LIN {X 0,Y 123.721,Z 466.518,A -85,B 0,C 180,E1 5812.106,E2 5812.106} C_VEL
LIN {X 0,Y 125.333,Z 474.545,A -85,B 0,C 180,E1 5807.962,E2 5807.962} C_VEL
LIN {X 0,Y 127.051,Z 480.548,A -85,B 0,C 180,E1 5806.881,E2 5806.881} C_VEL
LIN {X 0,Y 126.719,Z 512.471,A -85,B 0,C 180,E1 5803.232,E2 5803.232} C_VEL
LIN {X 0,Y 126.942,Z 529.099,A -85,B 0,C 180,E1 5801.274,E2 5801.274} C_VEL
LIN {X 0,Y 116.275,Z 624.974,A -85,B 0,C 180,E1 5791.007,E2 5791.007} C_VEL
LIN {X 0,Y 114.11,Z 644.035,A -85,B 0,C 180,E1 5787.956,E2 5787.956} C_VEL
LIN {X 0,Y 111.654,Z 663.331,A -85,B 0,C 180,E1 5783.765,E2 5783.765} C_VEL
LIN {X 0,Y 109.356,Z 682.14,A -85,B 0,C 180,E1 5778.388,E2 5778.388} C_VEL
LIN {X 0,Y 107.675,Z 699.18,A -85,B 0,C 180,E1 5772.061,E2 5772.061} C_VEL
LIN {X 0,Y 106.977,Z 713.625,A -85,B 0,C 180,E1 5765.364,E2 5765.364} C_VEL
LIN {X 0,Y 107.37,Z 725.986,A -85,B 0,C 180,E1 5758.4,E2 5758.4} C_VEL
LIN {X 0,Y 109.143,Z 736.932,A -85,B 0,C 180,E1 5751.041,E2 5751.041} C_VEL
LIN {X 0,Y 113.112,Z 747.249,A -85,B 0,C 180,E1 5743.041,E2 5743.041} C_VEL
LIN {X 0,Y 119.26,Z 755.624,A -85,B 0,C 180,E1 5735.745,E2 5735.745} C_VEL
LIN {X 0,Y 127.977,Z 762.647,A -85,B 0,C 180,E1 5728.96,E2 5728.96} C_VEL
LIN {X 0,Y 139.113,Z 768.269,A -85,B 0,C 180,E1 5722.921,E2 5722.921} C_VEL
LIN {X 0,Y 124.03,Z 769.681,A -85,B 0,C 180,E1 5713.891,E2 5713.891} C_VEL
LIN {X 0,Y 113.887,Z 769.686,A -85,B 0,C 180,E1 5702.381,E2 5702.381} C_VEL
LIN {X 0,Y 110.648,Z 768.902,A -85,B 0,C 180,E1 5693.994,E2 5693.994} C_VEL
LIN {X 0,Y 107.857,Z 776.455,A -85,B 0,C 180,E1 5688.933,E2 5688.933} C_VEL
LIN {X 0,Y 106.873,Z 787.522,A -85,B 0,C 180,E1 5680.239,E2 5680.239} C_VEL
LIN {X 0,Y 107.326,Z 795.234,A -85,B 0,C 180,E1 5672.67,E2 5672.67} C_VEL
LIN {X 0,Y 107.583,Z 799.108,A -85,B 0,C 180,E1 5667.87,E2 5667.87} C_VEL
LIN {X 0,Y 106.675,Z 803.029,A -85,B 0,C 180,E1 5660.831,E2 5660.831} C_VEL
LIN {X 0,Y 107.675,Z 807.586,A -85,B 0,C 180,E1 5649.337,E2 5649.337} C_VEL
LIN {X 0,Y 113.967,Z 810.858,A -85,B 0,C 180,E1 5637.048,E2 5637.048} C_VEL
LIN {X 0,Y 126.113,Z 812.492,A -85,B 0,C 180,E1 5626.176,E2 5626.176} C_VEL
LIN {X 0,Y 126.877,Z 812.523,A -85,B 0,C 180,E1 5625.679,E2 5625.679} C_VEL
LIN {X 0,Y 127.463,Z 812.423,A -85,B 0,C 180,E1 5624.581,E2 5624.581} C_VEL
LIN {X 0,Y 126.538,Z 812.035,A -85,B 0,C 180,E1 5623.133,E2 5623.133} C_VEL
LIN {X 0,Y 123.586,Z 811.164,A -85,B 0,C 180,E1 5621.271,E2 5621.271} C_VEL
LIN {X 0,Y 114.796,Z 808.547,A -85,B 0,C 180,E1 5617.036,E2 5617.036} C_VEL
LIN {X 0,Y 113.804,Z 808.153,A -85,B 0,C 180,E1 5616.3,E2 5616.3} C_VEL
LIN {X 0,Y 103.814,Z 802.035,A -85,B 0,C 180,E1 5605.072,E2 5605.072} C_VEL
LIN {X 0,Y 98.87,Z 794.82,A -85,B 0,C 180,E1 5593.449,E2 5593.449} C_VEL
LIN {X 0,Y 97.448,Z 787.451,A -85,B 0,C 180,E1 5583.529,E2 5583.529} C_VEL
LIN {X 0,Y 97.238,Z 779.92,A -85,B 0,C 180,E1 5575.281,E2 5575.281} C_VEL
LIN {X 0,Y 98.022,Z 769.975,A -85,B 0,C 180,E1 5566.431,E2 5566.431} C_VEL
LIN {X 0,Y 100.32,Z 757.927,A -85,B 0,C 180,E1 5557.744,E2 5557.744} C_VEL
LIN {X 0,Y 104.103,Z 744.078,A -85,B 0,C 180,E1 5549.815,E2 5549.815} C_VEL
LIN {X 0,Y 109.128,Z 728.223,A -85,B 0,C 180,E1 5542.791,E2 5542.791} C_VEL
LIN {X 0,Y 114.606,Z 711.516,A -85,B 0,C 180,E1 5537.116,E2 5537.116} C_VEL
LIN {X 0,Y 120.618,Z 692.425,A -85,B 0,C 180,E1 5532.179,E2 5532.179} C_VEL
LIN {X 0,Y 125.944,Z 673.888,A -85,B 0,C 180,E1 5528.557,E2 5528.557} C_VEL
LIN {X 0,Y 131.132,Z 652.804,A -85,B 0,C 180,E1 5525.515,E2 5525.515} C_VEL
LIN {X 0,Y 135.576,Z 630.555,A -85,B 0,C 180,E1 5523.193,E2 5523.193} C_VEL
LIN {X 0,Y 155.35,Z 515.756,A -85,B 0,C 180,E1 5515.036,E2 5515.036} C_VEL
LIN {X 0,Y 146.72,Z 495.36,A -85,B 0,C 180,E1 5509.751,E2 5509.751} C_VEL
LIN {X 0,Y 139.149,Z 478.944,A -85,B 0,C 180,E1 5504.513,E2 5504.513} C_VEL
LIN {X 0,Y 132.05,Z 464.915,A -85,B 0,C 180,E1 5498.93,E2 5498.93} C_VEL
LIN {X 0,Y 126.321,Z 454.594,A -85,B 0,C 180,E1 5493.79,E2 5493.79} C_VEL
LIN {X 0,Y 121.035,Z 445.893,A -85,B 0,C 180,E1 5488.344,E2 5488.344} C_VEL
LIN {X 0,Y 117.879,Z 441.07,A -85,B 0,C 180,E1 5484.646,E2 5484.646} C_VEL
LIN {X 0,Y 115.952,Z 438.032,A -85,B 0,C 180,E1 5482.07,E2 5482.07} C_VEL
LIN {X 0,Y 112.145,Z 438.158,A -85,B 0,C 180,E1 5478.167,E2 5478.167} C_VEL
LIN {X 0,Y 109.969,Z 438.898,A -85,B 0,C 180,E1 5475.789,E2 5475.789} C_VEL
LIN {X 0,Y 108.87,Z 438.667,A -85,B 0,C 180,E1 5474.28,E2 5474.28} C_VEL
LIN {X 0,Y 111.114,Z 446.42,A -85,B 0,C 180,E1 5467.794,E2 5467.794} C_VEL
LIN {X 0,Y 113.434,Z 455.846,A -85,B 0,C 180,E1 5461.001,E2 5461.001} C_VEL
LIN {X 0,Y 115.802,Z 466.855,A -85,B 0,C 180,E1 5454.046,E2 5454.046} C_VEL
LIN {X 0,Y 117.31,Z 474.41,A -85,B 0,C 180,E1 5449.866,E2 5449.866} C_VEL
LIN {X 0,Y 119.728,Z 482.332,A -85,B 0,C 180,E1 5448.282,E2 5448.282} C_VEL
LIN {X 0,Y 119.282,Z 515.284,A -85,B 0,C 180,E1 5444.26,E2 5444.26} C_VEL
LIN {X 0,Y 119.355,Z 529.39,A -85,B 0,C 180,E1 5442.498,E2 5442.498} C_VEL
LIN {X 0,Y 108.536,Z 622.949,A -85,B 0,C 180,E1 5431.831,E2 5431.831} C_VEL
LIN {X 0,Y 106.255,Z 642.844,A -85,B 0,C 180,E1 5428.527,E2 5428.527} C_VEL
LIN {X 0,Y 103.774,Z 662.039,A -85,B 0,C 180,E1 5424.173,E2 5424.173} C_VEL
LIN {X 0,Y 101.618,Z 679.408,A -85,B 0,C 180,E1 5418.948,E2 5418.948} C_VEL
LIN {X 0,Y 99.948,Z 695.818,A -85,B 0,C 180,E1 5412.715,E2 5412.715} C_VEL
LIN {X 0,Y 99.177,Z 710.919,A -85,B 0,C 180,E1 5405.497,E2 5405.497} C_VEL
LIN {X 0,Y 99.552,Z 723.373,A -85,B 0,C 180,E1 5398.274,E2 5398.274} C_VEL
LIN {X 0,Y 101.704,Z 736.139,A -85,B 0,C 180,E1 5389.457,E2 5389.457} C_VEL
LIN {X 0,Y 106.251,Z 746.98,A -85,B 0,C 180,E1 5380.771,E2 5380.771} C_VEL
LIN {X 0,Y 113.993,Z 756.585,A -85,B 0,C 180,E1 5372.299,E2 5372.299} C_VEL
LIN {X 0,Y 123.628,Z 763.772,A -85,B 0,C 180,E1 5365.52,E2 5365.52} C_VEL
LIN {X 0,Y 128.584,Z 766.518,A -85,B 0,C 180,E1 5362.772,E2 5362.772} C_VEL
LIN {X 0,Y 114.403,Z 766.985,A -85,B 0,C 180,E1 5352.977,E2 5352.977} C_VEL
LIN {X 0,Y 105.299,Z 766.112,A -85,B 0,C 180,E1 5340.216,E2 5340.216} C_VEL
LIN {X 0,Y 103.59,Z 765.612,A -85,B 0,C 180,E1 5335.131,E2 5335.131} C_VEL
LIN {X 0,Y 100.37,Z 773.329,A -85,B 0,C 180,E1 5329.798,E2 5329.798} C_VEL
LIN {X 0,Y 99.169,Z 784.781,A -85,B 0,C 180,E1 5320.456,E2 5320.456} C_VEL
LIN {X 0,Y 99.688,Z 792.768,A -85,B 0,C 180,E1 5312.299,E2 5312.299} C_VEL
LIN {X 0,Y 100.047,Z 796.404,A -85,B 0,C 180,E1 5307.709,E2 5307.709} C_VEL
LIN {X 0,Y 99.083,Z 800.833,A -85,B 0,C 180,E1 5299.535,E2 5299.535} C_VEL
LIN {X 0,Y 100.78,Z 805.742,A -85,B 0,C 180,E1 5286.619,E2 5286.619} C_VEL
LIN {X 0,Y 108.267,Z 809.203,A -85,B 0,C 180,E1 5273.768,E2 5273.768} C_VEL
LIN {X 0,Y 121.516,Z 811.112,A -85,B 0,C 180,E1 5262.919,E2 5262.919} C_VEL
LIN {X 0,Y 122.391,Z 811.157,A -85,B 0,C 180,E1 5262.319,E2 5262.319} C_VEL
LIN {X 0,Y 113.804,Z 808.153,A -85,B 0,C 180,E1 5256.3,E2 5256.3} C_VEL
LIN {X 0,Y 109.274,Z 806.262,A -85,B 0,C 180,E1 5253.207,E2 5253.207} C_VEL
LIN {X 0,Y 96.639,Z 799.888,A -85,B 0,C 180,E1 5245.209,E2 5245.209} C_VEL
LIN {X 0,Y 93.598,Z 797.166,A -85,B 0,C 180,E1 5241.222,E2 5241.222} C_VEL
LIN {X 0,Y 90.215,Z 789.137,A -85,B 0,C 180,E1 5228.925,E2 5228.925} C_VEL
LIN {X 0,Y 89.552,Z 782.607,A -85,B 0,C 180,E1 5220.639,E2 5220.639} C_VEL
LIN {X 0,Y 89.61,Z 774.104,A -85,B 0,C 180,E1 5211.659,E2 5211.659} C_VEL
LIN {X 0,Y 91.062,Z 762.989,A -85,B 0,C 180,E1 5202.094,E2 5202.094} C_VEL
LIN {X 0,Y 94.319,Z 749.505,A -85,B 0,C 180,E1 5192.881,E2 5192.881} C_VEL
LIN {X 0,Y 99.036,Z 734.325,A -85,B 0,C 180,E1 5184.863,E2 5184.863} C_VEL
LIN {X 0,Y 104.744,Z 717.443,A -85,B 0,C 180,E1 5178.07,E2 5178.07} C_VEL
LIN {X 0,Y 110.762,Z 699.456,A -85,B 0,C 180,E1 5172.612,E2 5172.612} C_VEL
LIN {X 0,Y 116.626,Z 680.494,A -85,B 0,C 180,E1 5168.329,E2 5168.329} C_VEL
LIN {X 0,Y 122.369,Z 659.306,A -85,B 0,C 180,E1 5164.797,E2 5164.797} C_VEL
LIN {X 0,Y 127.131,Z 637.978,A -85,B 0,C 180,E1 5162.224,E2 5162.224} C_VEL
LIN {X 0,Y 145.128,Z 537.776,A -85,B 0,C 180,E1 5154.544,E2 5154.544} C_VEL
LIN {X 0,Y 148.695,Z 518.047,A -85,B 0,C 180,E1 5153.269,E2 5153.269} C_VEL
LIN {X 0,Y 140.634,Z 498.608,A -85,B 0,C 180,E1 5147.908,E2 5147.908} C_VEL
LIN {X 0,Y 133.872,Z 483.562,A -85,B 0,C 180,E1 5142.838,E2 5142.838} C_VEL
LIN {X 0,Y 127.212,Z 469.981,A -85,B 0,C 180,E1 5137.162,E2 5137.162} C_VEL
LIN {X 0,Y 121.883,Z 460.1,A -85,B 0,C 180,E1 5131.946,E2 5131.946} C_VEL
LIN {X 0,Y 117.073,Z 451.938,A -85,B 0,C 180,E1 5126.573,E2 5126.573} C_VEL
LIN {X 0,Y 114.17,Z 447.292,A -85,B 0,C 180,E1 5122.831,E2 5122.831} C_VEL
LIN {X 0,Y 113.07,Z 445.717,A -85,B 0,C 180,E1 5121.354,E2 5121.354} C_VEL
LIN {X 0,Y 110.544,Z 446.078,A -85,B 0,C 180,E1 5118.786,E2 5118.786} C_VEL
LIN {X 0,Y 107.633,Z 446.625,A -85,B 0,C 180,E1 5115.474,E2 5115.474} C_VEL
LIN {X 0,Y 104.899,Z 448.123,A -85,B 0,C 180,E1 5112.241,E2 5112.241} C_VEL
LIN {X 0,Y 103.67,Z 448.229,A -85,B 0,C 180,E1 5110.124,E2 5110.124} C_VEL
LIN {X 0,Y 105.846,Z 457.247,A -85,B 0,C 180,E1 5103.036,E2 5103.036} C_VEL
LIN {X 0,Y 108.015,Z 467.637,A -85,B 0,C 180,E1 5095.942,E2 5095.942} C_VEL
LIN {X 0,Y 109.337,Z 474.358,A -85,B 0,C 180,E1 5091.966,E2 5091.966} C_VEL
LIN {X 0,Y 112.418,Z 484.295,A -85,B 0,C 180,E1 5089.775,E2 5089.775} C_VEL
LIN {X 0,Y 111.853,Z 518.434,A -85,B 0,C 180,E1 5085.323,E2 5085.323} C_VEL
LIN {X 0,Y 111.808,Z 529.579,A -85,B 0,C 180,E1 5083.851,E2 5083.851} C_VEL
LIN {X 0,Y 100.23,Z 626.422,A -85,B 0,C 180,E1 5071.919,E2 5071.919} C_VEL
LIN {X 0,Y 97.916,Z 645.376,A -85,B 0,C 180,E1 5068.349,E2 5068.349} C_VEL
LIN {X 0,Y 95.286,Z 665.471,A -85,B 0,C 180,E1 5063.173,E2 5063.173} C_VEL
LIN {X 0,Y 93.159,Z 683.027,A -85,B 0,C 180,E1 5057.209,E2 5057.209} C_VEL
LIN {X 0,Y 91.742,Z 699.415,A -85,B 0,C 180,E1 5050.043,E2 5050.043} C_VEL
LIN {X 0,Y 91.405,Z 712.924,A -85,B 0,C 180,E1 5042.822,E2 5042.822} C_VEL
LIN {X 0,Y 92.524,Z 726.836,A -85,B 0,C 180,E1 5033.797,E2 5033.797} C_VEL
LIN {X 0,Y 95.591,Z 738.612,A -85,B 0,C 180,E1 5024.842,E2 5024.842} C_VEL
LIN {X 0,Y 102.11,Z 750.1,A -85,B 0,C 180,E1 5015.1,E2 5015.1} C_VEL
LIN {X 0,Y 111.506,Z 759.323,A -85,B 0,C 180,E1 5006.841,E2 5006.841} C_VEL
LIN {X 0,Y 118.345,Z 763.963,A -85,B 0,C 180,E1 5002.534,E2 5002.534} C_VEL
LIN {X 0,Y 104.148,Z 763.568,A -85,B 0,C 180,E1 4990.755,E2 4990.755} C_VEL
LIN {X 0,Y 96.875,Z 761.886,A -85,B 0,C 180,E1 4976.678,E2 4976.678} C_VEL
LIN {X 0,Y 93.002,Z 769.991,A -85,B 0,C 180,E1 4970.78,E2 4970.78} C_VEL
LIN {X 0,Y 91.512,Z 782.027,A -85,B 0,C 180,E1 4960.478,E2 4960.478} C_VEL
LIN {X 0,Y 92.092,Z 790.143,A -85,B 0,C 180,E1 4951.867,E2 4951.867} C_VEL
LIN {X 0,Y 92.515,Z 793.931,A -85,B 0,C 180,E1 4946.902,E2 4946.902} C_VEL
LIN {X 0,Y 91.623,Z 798.409,A -85,B 0,C 180,E1 4938.033,E2 4938.033} C_VEL
LIN {X 0,Y 93.946,Z 803.567,A -85,B 0,C 180,E1 4924.128,E2 4924.128} C_VEL
LIN {X 0,Y 102.499,Z 807.357,A -85,B 0,C 180,E1 4910.649,E2 4910.649} C_VEL
LIN {X 0,Y 112.424,Z 809.109,A -85,B 0,C 180,E1 4902.424,E2 4902.424} C_VEL
LIN {X 0,Y 99.893,Z 803.047,A -85,B 0,C 180,E1 4891.364,E2 4891.364} C_VEL
LIN {X 0,Y 93.598,Z 797.166,A -85,B 0,C 180,E1 4881.222,E2 4881.222} C_VEL
LIN {X 0,Y 91.082,Z 794.298,A -85,B 0,C 180,E1 4877.067,E2 4877.067} C_VEL
LIN {X 0,Y 85.995,Z 788.825,A -85,B 0,C 180,E1 4870.746,E2 4870.746} C_VEL
LIN {X 0,Y 82.222,Z 782.653,A -85,B 0,C 180,E1 4863.824,E2 4863.824} C_VEL
LIN {X 0,Y 81.888,Z 780.974,A -85,B 0,C 180,E1 4861.77,E2 4861.77} C_VEL
LIN {X 0,Y 81.828,Z 772.489,A -85,B 0,C 180,E1 4852.275,E2 4852.275} C_VEL
LIN {X 0,Y 83.277,Z 761.101,A -85,B 0,C 180,E1 4841.809,E2 4841.809} C_VEL
LIN {X 0,Y 86.73,Z 747.302,A -85,B 0,C 180,E1 4831.792,E2 4831.792} C_VEL
LIN {X 0,Y 91.77,Z 731.804,A -85,B 0,C 180,E1 4823.183,E2 4823.183} C_VEL
LIN {X 0,Y 97.734,Z 714.838,A -85,B 0,C 180,E1 4816.143,E2 4816.143} C_VEL
LIN {X 0,Y 103.978,Z 696.725,A -85,B 0,C 180,E1 4810.564,E2 4810.564} C_VEL
LIN {X 0,Y 110.169,Z 677.178,A -85,B 0,C 180,E1 4806.124,E2 4806.124} C_VEL
LIN {X 0,Y 115.848,Z 656.61,A -85,B 0,C 180,E1 4802.699,E2 4802.699} C_VEL
LIN {X 0,Y 120.749,Z 634.715,A -85,B 0,C 180,E1 4800.11,E2 4800.11} C_VEL
LIN {X 0,Y 142.151,Z 520.396,A -85,B 0,C 180,E1 4791.4,E2 4791.4} C_VEL
LIN {X 0,Y 134.468,Z 501.434,A -85,B 0,C 180,E1 4785.803,E2 4785.803} C_VEL
LIN {X 0,Y 127.943,Z 486.588,A -85,B 0,C 180,E1 4780.429,E2 4780.429} C_VEL
LIN {X 0,Y 121.851,Z 473.881,A -85,B 0,C 180,E1 4774.707,E2 4774.707} C_VEL
LIN {X 0,Y 116.348,Z 463.379,A -85,B 0,C 180,E1 4768.646,E2 4768.646} C_VEL
LIN {X 0,Y 111.637,Z 455.203,A -85,B 0,C 180,E1 4762.538,E2 4762.538} C_VEL
LIN {X 0,Y 110.391,Z 453.587,A -85,B 0,C 180,E1 4760.849,E2 4760.849} C_VEL
LIN {X 0,Y 105.65,Z 454.774,A -85,B 0,C 180,E1 4755.755,E2 4755.755} C_VEL
LIN {X 0,Y 102.852,Z 455.957,A -85,B 0,C 180,E1 4752.308,E2 4752.308} C_VEL
LIN {X 0,Y 101.988,Z 456.324,A -85,B 0,C 180,E1 4751.124,E2 4751.124} C_VEL
LIN {X 0,Y 99.384,Z 458.401,A -85,B 0,C 180,E1 4747.523,E2 4747.523} C_VEL
LIN {X 0,Y 98.286,Z 458.631,A -85,B 0,C 180,E1 4745.349,E2 4745.349} C_VEL
LIN {X 0,Y 100.3,Z 468.623,A -85,B 0,C 180,E1 4737.925,E2 4737.925} C_VEL
LIN {X 0,Y 101.387,Z 474.232,A -85,B 0,C 180,E1 4734.332,E2 4734.332} C_VEL
LIN {X 0,Y 105.158,Z 486.038,A -85,B 0,C 180,E1 4731.45,E2 4731.45} C_VEL
LIN {X 0,Y 104.426,Z 521.241,A -85,B 0,C 180,E1 4726.525,E2 4726.525} C_VEL
LIN {X 0,Y 104.26,Z 529.903,A -85,B 0,C 180,E1 4725.316,E2 4725.316} C_VEL
LIN {X 0,Y 92.313,Z 625.986,A -85,B 0,C 180,E1 4712.56,E2 4712.56} C_VEL
LIN {X 0,Y 89.751,Z 646.386,A -85,B 0,C 180,E1 4708.41,E2 4708.41} C_VEL
LIN {X 0,Y 87.193,Z 665.725,A -85,B 0,C 180,E1 4702.948,E2 4702.948} C_VEL
LIN {X 0,Y 85.022,Z 684.07,A -85,B 0,C 180,E1 4696.044,E2 4696.044} C_VEL
LIN {X 0,Y 83.846,Z 699.623,A -85,B 0,C 180,E1 4688.573,E2 4688.573} C_VEL
LIN {X 0,Y 83.83,Z 714.169,A -85,B 0,C 180,E1 4680.001,E2 4680.001} C_VEL
LIN {X 0,Y 85.319,Z 726.551,A -85,B 0,C 180,E1 4671.238,E2 4671.238} C_VEL
LIN {X 0,Y 89.029,Z 738.457,A -85,B 0,C 180,E1 4661.673,E2 4661.673} C_VEL
LIN {X 0,Y 95.494,Z 748.999,A -85,B 0,C 180,E1 4652.569,E2 4652.569} C_VEL
LIN {X 0,Y 104.93,Z 758.162,A -85,B 0,C 180,E1 4644.462,E2 4644.462} C_VEL
LIN {X 0,Y 108.323,Z 760.799,A -85,B 0,C 180,E1 4642.111,E2 4642.111} C_VEL
LIN {X 0,Y 95.171,Z 759.575,A -85,B 0,C 180,E1 4629.077,E2 4629.077} C_VEL
LIN {X 0,Y 90.239,Z 758.073,A -85,B 0,C 180,E1 4618.273,E2 4618.273} C_VEL
LIN {X 0,Y 86.024,Z 765.743,A -85,B 0,C 180,E1 4612.554,E2 4612.554} C_VEL
LIN {X 0,Y 83.939,Z 776.554,A -85,B 0,C 180,E1 4603.081,E2 4603.081} C_VEL
LIN {X 0,Y 84.274,Z 785.664,A -85,B 0,C 180,E1 4593.401,E2 4593.401} C_VEL
LIN {X 0,Y 85.113,Z 790.885,A -85,B 0,C 180,E1 4586.633,E2 4586.633} C_VEL
LIN {X 0,Y 84.257,Z 795.604,A -85,B 0,C 180,E1 4576.969,E2 4576.969} C_VEL
LIN {X 0,Y 87.097,Z 801.024,A -85,B 0,C 180,E1 4561.922,E2 4561.922} C_VEL
LIN {X 0,Y 97.124,Z 805.268,A -85,B 0,C 180,E1 4547.199,E2 4547.199} C_VEL
LIN {X 0,Y 102.565,Z 806.461,A -85,B 0,C 180,E1 4542.46,E2 4542.46} C_VEL
LIN {X 0,Y 90.222,Z 799.306,A -85,B 0,C 180,E1 4529.913,E2 4529.913} C_VEL
LIN {X 0,Y 83.846,Z 790.967,A -85,B 0,C 180,E1 4515.918,E2 4515.918} C_VEL
LIN {X 0,Y 82.11,Z 783.382,A -85,B 0,C 180,E1 4504.889,E2 4504.889} C_VEL
LIN {X 0,Y 81.888,Z 780.974,A -85,B 0,C 180,E1 4501.77,E2 4501.77} C_VEL
LIN {X 0,Y 81.018,Z 777.486,A -85,B 0,C 180,E1 4497.857,E2 4497.857} C_VEL
LIN {X 0,Y 78.361,Z 771.552,A -85,B 0,C 180,E1 4492.363,E2 4492.363} C_VEL
LIN {X 0,Y 75.4,Z 762.922,A -85,B 0,C 180,E1 4484.847,E2 4484.847} C_VEL
LIN {X 0,Y 75.493,Z 759.219,A -85,B 0,C 180,E1 4481.571,E2 4481.571} C_VEL
LIN {X 0,Y 78.882,Z 745.991,A -85,B 0,C 180,E1 4471.205,E2 4471.205} C_VEL
LIN {X 0,Y 84.18,Z 730.279,A -85,B 0,C 180,E1 4461.855,E2 4461.855} C_VEL
LIN {X 0,Y 90.363,Z 713.341,A -85,B 0,C 180,E1 4454.463,E2 4454.463} C_VEL
LIN {X 0,Y 97.067,Z 694.602,A -85,B 0,C 180,E1 4448.476,E2 4448.476} C_VEL
LIN {X 0,Y 103.57,Z 674.696,A -85,B 0,C 180,E1 4443.875,E2 4443.875} C_VEL
LIN {X 0,Y 109.519,Z 653.453,A -85,B 0,C 180,E1 4440.373,E2 4440.373} C_VEL
LIN {X 0,Y 114.494,Z 631.417,A -85,B 0,C 180,E1 4437.811,E2 4437.811} C_VEL
LIN {X 0,Y 135.589,Z 522.526,A -85,B 0,C 180,E1 4429.324,E2 4429.324} C_VEL
LIN {X 0,Y 128.396,Z 504.331,A -85,B 0,C 180,E1 4423.573,E2 4423.573} C_VEL
LIN {X 0,Y 122.113,Z 489.542,A -85,B 0,C 180,E1 4417.796,E2 4417.796} C_VEL
LIN {X 0,Y 116.23,Z 476.958,A -85,B 0,C 180,E1 4411.602,E2 4411.602} C_VEL
LIN {X 0,Y 110.768,Z 466.31,A -85,B 0,C 180,E1 4404.691,E2 4404.691} C_VEL
LIN {X 0,Y 108.029,Z 461.515,A -85,B 0,C 180,E1 4400.679,E2 4400.679} C_VEL
LIN {X 0,Y 104.264,Z 462.552,A -85,B 0,C 180,E1 4396.694,E2 4396.694} C_VEL
LIN {X 0,Y 100.714,Z 464.062,A -85,B 0,C 180,E1 4392.378,E2 4392.378} C_VEL
LIN {X 0,Y 97.805,Z 466.095,A -85,B 0,C 180,E1 4388.406,E2 4388.406} C_VEL
LIN {X 0,Y 96.699,Z 466.726,A -85,B 0,C 180,E1 4386.589,E2 4386.589} C_VEL
LIN {X 0,Y 94.001,Z 469.898,A -85,B 0,C 180,E1 4382.249,E2 4382.249} C_VEL
LIN {X 0,Y 92.834,Z 470.83,A -85,B 0,C 180,E1 4379.23,E2 4379.23} C_VEL
LIN {X 0,Y 93.482,Z 474.123,A -85,B 0,C 180,E1 4377.033,E2 4377.033} C_VEL
LIN {X 0,Y 97.927,Z 487.871,A -85,B 0,C 180,E1 4373.276,E2 4373.276} C_VEL
LIN {X 0,Y 97.007,Z 524.973,A -85,B 0,C 180,E1 4367.689,E2 4367.689} C_VEL
LIN {X 0,Y 96.664,Z 530.708,A -85,B 0,C 180,E1 4366.877,E2 4366.877} C_VEL
LIN {X 0,Y 84.165,Z 627.528,A -85,B 0,C 180,E1 4352.898,E2 4352.898} C_VEL
LIN {X 0,Y 81.651,Z 646.801,A -85,B 0,C 180,E1 4348.528,E2 4348.528} C_VEL
LIN {X 0,Y 79.007,Z 666.672,A -85,B 0,C 180,E1 4342.313,E2 4342.313} C_VEL
LIN {X 0,Y 77.022,Z 684.046,A -85,B 0,C 180,E1 4335.049,E2 4335.049} C_VEL
LIN {X 0,Y 76.041,Z 699.625,A -85,B 0,C 180,E1 4326.797,E2 4326.797} C_VEL
LIN {X 0,Y 76.366,Z 713.602,A -85,B 0,C 180,E1 4317.75,E2 4317.75} C_VEL
LIN {X 0,Y 78.317,Z 726.203,A -85,B 0,C 180,E1 4308.214,E2 4308.214} C_VEL
LIN {X 0,Y 83.182,Z 738.924,A -85,B 0,C 180,E1 4297.379,E2 4297.379} C_VEL
LIN {X 0,Y 91.282,Z 750.114,A -85,B 0,C 180,E1 4287.54,E2 4287.54} C_VEL
LIN {X 0,Y 98.67,Z 756.927,A -85,B 0,C 180,E1 4281.541,E2 4281.541} C_VEL
LIN {X 0,Y 86.238,Z 754.891,A -85,B 0,C 180,E1 4266.25,E2 4266.25} C_VEL
LIN {X 0,Y 83.89,Z 753.99,A -85,B 0,C 180,E1 4260.236,E2 4260.236} C_VEL
LIN {X 0,Y 79.275,Z 761.328,A -85,B 0,C 180,E1 4254.596,E2 4254.596} C_VEL
LIN {X 0,Y 76.54,Z 770.847,A -85,B 0,C 180,E1 4245.922,E2 4245.922} C_VEL
LIN {X 0,Y 76.498,Z 780.779,A -85,B 0,C 180,E1 4235.25,E2 4235.25} C_VEL
LIN {X 0,Y 77.704,Z 787.693,A -85,B 0,C 180,E1 4226.311,E2 4226.311} C_VEL
LIN {X 0,Y 77.01,Z 791.977,A -85,B 0,C 180,E1 4217.249,E2 4217.249} C_VEL
LIN {X 0,Y 79.877,Z 797.867,A -85,B 0,C 180,E1 4200.779,E2 4200.779} C_VEL
LIN {X 0,Y 90.361,Z 802.559,A -85,B 0,C 180,E1 4185.085,E2 4185.085} C_VEL
LIN {X 0,Y 92.988,Z 803.281,A -85,B 0,C 180,E1 4182.641,E2 4182.641} C_VEL
LIN {X 0,Y 81.109,Z 795.266,A -85,B 0,C 180,E1 4168.735,E2 4168.735} C_VEL
LIN {X 0,Y 75.617,Z 786.418,A -85,B 0,C 180,E1 4153.768,E2 4153.768} C_VEL
LIN {X 0,Y 74.306,Z 778.93,A -85,B 0,C 180,E1 4142.893,E2 4142.893} C_VEL
LIN {X 0,Y 74.079,Z 770.779,A -85,B 0,C 180,E1 4133.022,E2 4133.022} C_VEL
LIN {X 0,Y 75.493,Z 759.219,A -85,B 0,C 180,E1 4121.571,E2 4121.571} C_VEL
LIN {X 0,Y 75.65,Z 753.984,A -85,B 0,C 180,E1 4117.24,E2 4117.24} C_VEL
LIN {X 0,Y 74.166,Z 744.301,A -85,B 0,C 180,E1 4110.222,E2 4110.222} C_VEL
LIN {X 0,Y 74.076,Z 736.656,A -85,B 0,C 180,E1 4105.087,E2 4105.087} C_VEL
LIN {X 0,Y 74.941,Z 733.22,A -85,B 0,C 180,E1 4102.951,E2 4102.951} C_VEL
LIN {X 0,Y 81.259,Z 716.528,A -85,B 0,C 180,E1 4094.464,E2 4094.464} C_VEL
LIN {X 0,Y 88.1,Z 698.388,A -85,B 0,C 180,E1 4087.876,E2 4087.876} C_VEL
LIN {X 0,Y 95.059,Z 678.413,A -85,B 0,C 180,E1 4082.703,E2 4082.703} C_VEL
LIN {X 0,Y 101.268,Z 657.994,A -85,B 0,C 180,E1 4078.934,E2 4078.934} C_VEL
LIN {X 0,Y 106.692,Z 635.926,A -85,B 0,C 180,E1 4076.113,E2 4076.113} C_VEL
LIN {X 0,Y 129.29,Z 525.084,A -85,B 0,C 180,E1 4067.206,E2 4067.206} C_VEL
LIN {X 0,Y 122.453,Z 507.2,A -85,B 0,C 180,E1 4061.17,E2 4061.17} C_VEL
LIN {X 0,Y 116.584,Z 492.994,A -85,B 0,C 180,E1 4055.142,E2 4055.142} C_VEL
LIN {X 0,Y 111.623,Z 481.965,A -85,B 0,C 180,E1 4049.294,E2 4049.294} C_VEL
LIN {X 0,Y 107.035,Z 472.552,A -85,B 0,C 180,E1 4042.89,E2 4042.89} C_VEL
LIN {X 0,Y 105.47,Z 469.603,A -85,B 0,C 180,E1 4040.378,E2 4040.378} C_VEL
LIN {X 0,Y 102.881,Z 470.299,A -85,B 0,C 180,E1 4037.654,E2 4037.654} C_VEL
LIN {X 0,Y 99.296,Z 471.895,A -85,B 0,C 180,E1 4033.458,E2 4033.458} C_VEL
LIN {X 0,Y 95.383,Z 474.453,A -85,B 0,C 180,E1 4028.082,E2 4028.082} C_VEL
LIN {X 0,Y 92.384,Z 477.586,A -85,B 0,C 180,E1 4023.311,E2 4023.311} C_VEL
LIN {X 0,Y 91.234,Z 478.654,A -85,B 0,C 180,E1 4020.929,E2 4020.929} C_VEL
LIN {X 0,Y 89.394,Z 482.633,A -85,B 0,C 180,E1 4018.219,E2 4018.219} C_VEL
LIN {X 0,Y 88.994,Z 483.763,A -85,B 0,C 180,E1 4017.029,E2 4017.029} C_VEL
LIN {X 0,Y 90.735,Z 490.079,A -85,B 0,C 180,E1 4015.279,E2 4015.279} C_VEL
LIN {X 0,Y 89.331,Z 530.129,A -85,B 0,C 180,E1 4008.818,E2 4008.818} C_VEL
LIN {X 0,Y 76.063,Z 628.474,A -85,B 0,C 180,E1 3993.306,E2 3993.306} C_VEL
LIN {X 0,Y 73.465,Z 647.791,A -85,B 0,C 180,E1 3988.449,E2 3988.449} C_VEL
LIN {X 0,Y 70.861,Z 667.353,A -85,B 0,C 180,E1 3981.523,E2 3981.523} C_VEL
LIN {X 0,Y 68.89,Z 686.196,A -85,B 0,C 180,E1 3972.576,E2 3972.576} C_VEL
LIN {X 0,Y 68.368,Z 701.323,A -85,B 0,C 180,E1 3963.355,E2 3963.355} C_VEL
LIN {X 0,Y 69.404,Z 715.573,A -85,B 0,C 180,E1 3952.967,E2 3952.967} C_VEL
LIN {X 0,Y 72.796,Z 729.076,A -85,B 0,C 180,E1 3941.586,E2 3941.586} C_VEL
LIN {X 0,Y 79.827,Z 742.098,A -85,B 0,C 180,E1 3929.934,E2 3929.934} C_VEL
LIN {X 0,Y 89.383,Z 752.538,A -85,B 0,C 180,E1 3920.773,E2 3920.773} C_VEL
LIN {X 0,Y 78.157,Z 749.724,A -85,B 0,C 180,E1 3903.374,E2 3903.374} C_VEL
LIN {X 0,Y 77.776,Z 749.693,A -85,B 0,C 180,E1 3902.461,E2 3902.461} C_VEL
LIN {X 0,Y 72.816,Z 756.642,A -85,B 0,C 180,E1 3896.945,E2 3896.945} C_VEL
LIN {X 0,Y 69.361,Z 765.595,A -85,B 0,C 180,E1 3888.49,E2 3888.49} C_VEL
LIN {X 0,Y 68.88,Z 776.874,A -85,B 0,C 180,E1 3875.832,E2 3875.832} C_VEL
LIN {X 0,Y 70.408,Z 784.699,A -85,B 0,C 180,E1 3865.112,E2 3865.112} C_VEL
LIN {X 0,Y 69.876,Z 789.052,A -85,B 0,C 180,E1 3855.074,E2 3855.074} C_VEL
LIN {X 0,Y 74.075,Z 795.388,A -85,B 0,C 180,E1 3836.398,E2 3836.398} C_VEL
LIN {X 0,Y 83.542,Z 799.491,A -85,B 0,C 180,E1 3822.804,E2 3822.804} C_VEL
LIN {X 0,Y 72.511,Z 791.042,A -85,B 0,C 180,E1 3807.957,E2 3807.957} C_VEL
LIN {X 0,Y 67.808,Z 782.318,A -85,B 0,C 180,E1 3792.777,E2 3792.777} C_VEL
LIN {X 0,Y 66.659,Z 775.559,A -85,B 0,C 180,E1 3782.578,E2 3782.578} C_VEL
LIN {X 0,Y 66.484,Z 766.656,A -85,B 0,C 180,E1 3771.349,E2 3771.349} C_VEL
LIN {X 0,Y 68.382,Z 754.22,A -85,B 0,C 180,E1 3758.558,E2 3758.558} C_VEL
LIN {X 0,Y 72.634,Z 739.743,A -85,B 0,C 180,E1 3747.11,E2 3747.11} C_VEL
LIN {X 0,Y 74.941,Z 733.22,A -85,B 0,C 180,E1 3742.951,E2 3742.951} C_VEL
LIN {X 0,Y 76.193,Z 727.143,A -85,B 0,C 180,E1 3739.421,E2 3739.421} C_VEL
LIN {X 0,Y 76.383,Z 713.469,A -85,B 0,C 180,E1 3732.091,E2 3732.091} C_VEL
LIN {X 0,Y 77.636,Z 705.905,A -85,B 0,C 180,E1 3728.659,E2 3728.659} C_VEL
LIN {X 0,Y 78.297,Z 703.986,A -85,B 0,C 180,E1 3727.928,E2 3727.928} C_VEL
LIN {X 0,Y 85.53,Z 684.851,A -85,B 0,C 180,E1 3722.054,E2 3722.054} C_VEL
LIN {X 0,Y 92.154,Z 665.009,A -85,B 0,C 180,E1 3717.81,E2 3717.81} C_VEL
LIN {X 0,Y 98.137,Z 643.486,A -85,B 0,C 180,E1 3714.587,E2 3714.587} C_VEL
LIN {X 0,Y 105.014,Z 611.799,A -85,B 0,C 180,E1 3711.36,E2 3711.36} C_VEL
LIN {X 0,Y 122.943,Z 527.227,A -85,B 0,C 180,E1 3704.783,E2 3704.783} C_VEL
LIN {X 0,Y 116.417,Z 509.537,A -85,B 0,C 180,E1 3698.333,E2 3698.333} C_VEL
LIN {X 0,Y 110.885,Z 495.637,A -85,B 0,C 180,E1 3691.873,E2 3691.873} C_VEL
LIN {X 0,Y 106.366,Z 485.172,A -85,B 0,C 180,E1 3685.687,E2 3685.687} C_VEL
LIN {X 0,Y 102.71,Z 477.567,A -85,B 0,C 180,E1 3679.829,E2 3679.829} C_VEL
LIN {X 0,Y 98.152,Z 479.522,A -85,B 0,C 180,E1 3674.812,E2 3674.812} C_VEL
LIN {X 0,Y 94.295,Z 481.971,A -85,B 0,C 180,E1 3669.789,E2 3669.789} C_VEL
LIN {X 0,Y 90.848,Z 485.226,A -85,B 0,C 180,E1 3664.488,E2 3664.488} C_VEL
LIN {X 0,Y 90.279,Z 485.976,A -85,B 0,C 180,E1 3663.602,E2 3663.602} C_VEL
LIN {X 0,Y 88.23,Z 489.907,A -85,B 0,C 180,E1 3660.764,E2 3660.764} C_VEL
LIN {X 0,Y 86.957,Z 493.361,A -85,B 0,C 180,E1 3659.504,E2 3659.504} C_VEL
LIN {X 0,Y 83.896,Z 502.205,A -85,B 0,C 180,E1 3656.819,E2 3656.819} C_VEL
LIN {X 0,Y 82.806,Z 505.573,A -85,B 0,C 180,E1 3655.29,E2 3655.29} C_VEL
LIN {X 0,Y 81.955,Z 530.078,A -85,B 0,C 180,E1 3650.921,E2 3650.921} C_VEL
LIN {X 0,Y 68.112,Z 628.15,A -85,B 0,C 180,E1 3634.034,E2 3634.034} C_VEL
LIN {X 0,Y 65.329,Z 648.28,A -85,B 0,C 180,E1 3628.325,E2 3628.325} C_VEL
LIN {X 0,Y 62.747,Z 667.856,A -85,B 0,C 180,E1 3620.523,E2 3620.523} C_VEL
LIN {X 0,Y 61.119,Z 684.923,A -85,B 0,C 180,E1 3611.322,E2 3611.322} C_VEL
LIN {X 0,Y 60.852,Z 700.406,A -85,B 0,C 180,E1 3600.943,E2 3600.943} C_VEL
LIN {X 0,Y 62.578,Z 715.186,A -85,B 0,C 180,E1 3588.947,E2 3588.947} C_VEL
LIN {X 0,Y 66.739,Z 728.344,A -85,B 0,C 180,E1 3577.076,E2 3577.076} C_VEL
LIN {X 0,Y 73.824,Z 740.101,A -85,B 0,C 180,E1 3566.27,E2 3566.27} C_VEL
LIN {X 0,Y 80.515,Z 747.565,A -85,B 0,C 180,E1 3559.779,E2 3559.779} C_VEL
LIN {X 0,Y 72.1,Z 745.036,A -85,B 0,C 180,E1 3545.136,E2 3545.136} C_VEL
LIN {X 0,Y 66.629,Z 751.824,A -85,B 0,C 180,E1 3539.684,E2 3539.684} C_VEL
LIN {X 0,Y 62.101,Z 761.699,A -85,B 0,C 180,E1 3529.762,E2 3529.762} C_VEL
LIN {X 0,Y 61.456,Z 774.051,A -85,B 0,C 180,E1 3514.666,E2 3514.666} C_VEL
LIN {X 0,Y 63.206,Z 781.852,A -85,B 0,C 180,E1 3503.186,E2 3503.186} C_VEL
LIN {X 0,Y 63.698,Z 788.191,A -85,B 0,C 180,E1 3485.913,E2 3485.913} C_VEL
LIN {X 0,Y 72.144,Z 794.377,A -85,B 0,C 180,E1 3466.11,E2 3466.11} C_VEL
LIN {X 0,Y 74.33,Z 795.204,A -85,B 0,C 180,E1 3463.052,E2 3463.052} C_VEL
LIN {X 0,Y 63.698,Z 785.836,A -85,B 0,C 180,E1 3446.071,E2 3446.071} C_VEL
LIN {X 0,Y 59.936,Z 777.233,A -85,B 0,C 180,E1 3430.573,E2 3430.573} C_VEL
LIN {X 0,Y 58.872,Z 769.628,A -85,B 0,C 180,E1 3419.026,E2 3419.026} C_VEL
LIN {X 0,Y 59.232,Z 759.734,A -85,B 0,C 180,E1 3406.329,E2 3406.329} C_VEL
LIN {X 0,Y 62.19,Z 746.447,A -85,B 0,C 180,E1 3392.727,E2 3392.727} C_VEL
LIN {X 0,Y 67.466,Z 731.259,A -85,B 0,C 180,E1 3381.208,E2 3381.208} C_VEL
LIN {X 0,Y 74.159,Z 714.372,A -85,B 0,C 180,E1 3372.135,E2 3372.135} C_VEL
LIN {X 0,Y 78.297,Z 703.986,A -85,B 0,C 180,E1 3367.928,E2 3367.928} C_VEL
LIN {X 0,Y 79.961,Z 697.284,A -85,B 0,C 180,E1 3365.367,E2 3365.367} C_VEL
LIN {X 0,Y 81.208,Z 678.536,A -85,B 0,C 180,E1 3358.294,E2 3358.294} C_VEL
LIN {X 0,Y 82.686,Z 672.39,A -85,B 0,C 180,E1 3356.682,E2 3356.682} C_VEL
LIN {X 0,Y 89.32,Z 651.279,A -85,B 0,C 180,E1 3352.967,E2 3352.967} C_VEL
LIN {X 0,Y 95.072,Z 628.181,A -85,B 0,C 180,E1 3350.229,E2 3350.229} C_VEL
LIN {X 0,Y 116.803,Z 529.586,A -85,B 0,C 180,E1 3342.229,E2 3342.229} C_VEL
LIN {X 0,Y 110.764,Z 512.531,A -85,B 0,C 180,E1 3335.504,E2 3335.504} C_VEL
LIN {X 0,Y 105.881,Z 499.542,A -85,B 0,C 180,E1 3328.992,E2 3328.992} C_VEL
LIN {X 0,Y 101.951,Z 489.947,A -85,B 0,C 180,E1 3322.817,E2 3322.817} C_VEL
LIN {X 0,Y 100.11,Z 485.795,A -85,B 0,C 180,E1 3319.537,E2 3319.537} C_VEL
LIN {X 0,Y 96.698,Z 487.363,A -85,B 0,C 180,E1 3315.796,E2 3315.796} C_VEL
LIN {X 0,Y 93.309,Z 489.435,A -85,B 0,C 180,E1 3311.572,E2 3311.572} C_VEL
LIN {X 0,Y 89.618,Z 492.908,A -85,B 0,C 180,E1 3306.368,E2 3306.368} C_VEL
LIN {X 0,Y 87.98,Z 495.911,A -85,B 0,C 180,E1 3304.431,E2 3304.431} C_VEL
LIN {X 0,Y 84.341,Z 505.672,A -85,B 0,C 180,E1 3301.749,E2 3301.749} C_VEL
LIN {X 0,Y 82.822,Z 509.668,A -85,B 0,C 180,E1 3300.282,E2 3300.282} C_VEL
LIN {X 0,Y 78.469,Z 522.921,A -85,B 0,C 180,E1 3297.33,E2 3297.33} C_VEL
LIN {X 0,Y 75.773,Z 531.128,A -85,B 0,C 180,E1 3294.628,E2 3294.628} C_VEL
LIN {X 0,Y 72.538,Z 542.204,A -85,B 0,C 180,E1 3291.587,E2 3291.587} C_VEL
LIN {X 0,Y 59.811,Z 630.351,A -85,B 0,C 180,E1 3274.131,E2 3274.131} C_VEL
LIN {X 0,Y 57.207,Z 648.632,A -85,B 0,C 180,E1 3268.159,E2 3268.159} C_VEL
LIN {X 0,Y 54.627,Z 668.707,A -85,B 0,C 180,E1 3258.816,E2 3258.816} C_VEL
LIN {X 0,Y 53.288,Z 686.652,A -85,B 0,C 180,E1 3247.549,E2 3247.549} C_VEL
LIN {X 0,Y 53.84,Z 702.268,A -85,B 0,C 180,E1 3235.208,E2 3235.208} C_VEL
LIN {X 0,Y 56.447,Z 715.685,A -85,B 0,C 180,E1 3223.008,E2 3223.008} C_VEL
LIN {X 0,Y 62.153,Z 729.144,A -85,B 0,C 180,E1 3210.088,E2 3210.088} C_VEL
LIN {X 0,Y 71.721,Z 741.877,A -85,B 0,C 180,E1 3198.534,E2 3198.534} C_VEL
LIN {X 0,Y 71.822,Z 742.081,A -85,B 0,C 180,E1 3198.142,E2 3198.142} C_VEL
LIN {X 0,Y 66.485,Z 740.424,A -85,B 0,C 180,E1 3188.069,E2 3188.069} C_VEL
LIN {X 0,Y 60.158,Z 747.649,A -85,B 0,C 180,E1 3182.131,E2 3182.131} C_VEL
LIN {X 0,Y 55.261,Z 756.798,A -85,B 0,C 180,E1 3172.332,E2 3172.332} C_VEL
LIN {X 0,Y 53.835,Z 768.898,A -85,B 0,C 180,E1 3156.398,E2 3156.398} C_VEL
LIN {X 0,Y 55.82,Z 777.661,A -85,B 0,C 180,E1 3142.797,E2 3142.797} C_VEL
LIN {X 0,Y 56.093,Z 778.719,A -85,B 0,C 180,E1 3140.769,E2 3140.769} C_VEL
LIN {X 0,Y 57.61,Z 785.357,A -85,B 0,C 180,E1 3120.924,E2 3120.924} C_VEL
LIN {X 0,Y 65.486,Z 790.526,A -85,B 0,C 180,E1 3103.576,E2 3103.576} C_VEL
LIN {X 0,Y 55.68,Z 781.021,A -85,B 0,C 180,E1 3085.528,E2 3085.528} C_VEL
LIN {X 0,Y 52.498,Z 773.381,A -85,B 0,C 180,E1 3070.978,E2 3070.978} C_VEL
LIN {X 0,Y 51.264,Z 765.286,A -85,B 0,C 180,E1 3057.763,E2 3057.763} C_VEL
LIN {X 0,Y 52.121,Z 753.798,A -85,B 0,C 180,E1 3042.124,E2 3042.124} C_VEL
LIN {X 0,Y 56.162,Z 739.404,A -85,B 0,C 180,E1 3027.11,E2 3027.11} C_VEL
LIN {X 0,Y 62.52,Z 723.197,A -85,B 0,C 180,E1 3015.276,E2 3015.276} C_VEL
LIN {X 0,Y 69.8,Z 705.904,A -85,B 0,C 180,E1 3006.659,E2 3006.659} C_VEL
LIN {X 0,Y 77.482,Z 686.748,A -85,B 0,C 180,E1 3000.161,E2 3000.161} C_VEL
LIN {X 0,Y 82.686,Z 672.39,A -85,B 0,C 180,E1 2996.682,E2 2996.682} C_VEL
LIN {X 0,Y 84.208,Z 665.256,A -85,B 0,C 180,E1 2994.92,E2 2994.92} C_VEL
LIN {X 0,Y 84.886,Z 645.536,A -85,B 0,C 180,E1 2989.455,E2 2989.455} C_VEL
LIN {X 0,Y 86.002,Z 639.13,A -85,B 0,C 180,E1 2988.385,E2 2988.385} C_VEL
LIN {X 0,Y 108.111,Z 543.66,A -85,B 0,C 180,E1 2980.229,E2 2980.229} C_VEL
LIN {X 0,Y 110.748,Z 531.852,A -85,B 0,C 180,E1 2979.412,E2 2979.412} C_VEL
LIN {X 0,Y 105.427,Z 515.873,A -85,B 0,C 180,E1 2972.582,E2 2972.582} C_VEL
LIN {X 0,Y 100.943,Z 503.158,A -85,B 0,C 180,E1 2965.668,E2 2965.668} C_VEL
LIN {X 0,Y 97.48,Z 494.085,A -85,B 0,C 180,E1 2959.211,E2 2959.211} C_VEL
LIN {X 0,Y 92.655,Z 496.628,A -85,B 0,C 180,E1 2953.705,E2 2953.705} C_VEL
LIN {X 0,Y 89,Z 499.921,A -85,B 0,C 180,E1 2949.047,E2 2949.047} C_VEL
LIN {X 0,Y 84.56,Z 510.839,A -85,B 0,C 180,E1 2945.986,E2 2945.986} C_VEL
LIN {X 0,Y 83.462,Z 513.651,A -85,B 0,C 180,E1 2945.233,E2 2945.233} C_VEL
LIN {X 0,Y 78.775,Z 527.027,A -85,B 0,C 180,E1 2942.389,E2 2942.389} C_VEL
LIN {X 0,Y 76.131,Z 534.344,A -85,B 0,C 180,E1 2940.186,E2 2940.186} C_VEL
LIN {X 0,Y 72.612,Z 545.015,A -85,B 0,C 180,E1 2937.595,E2 2937.595} C_VEL
LIN {X 0,Y 62.799,Z 578.204,A -85,B 0,C 180,E1 2931.679,E2 2931.679} C_VEL
LIN {X 0,Y 57.177,Z 598.126,A -85,B 0,C 180,E1 2925.709,E2 2925.709} C_VEL
LIN {X 0,Y 54.55,Z 609.115,A -85,B 0,C 180,E1 2920.509,E2 2920.509} C_VEL
LIN {X 0,Y 51.161,Z 634.743,A -85,B 0,C 180,E1 2913.345,E2 2913.345} C_VEL
LIN {X 0,Y 48.328,Z 654.422,A -85,B 0,C 180,E1 2905.097,E2 2905.097} C_VEL
LIN {X 0,Y 46.457,Z 670.849,A -85,B 0,C 180,E1 2895.556,E2 2895.556} C_VEL
LIN {X 0,Y 45.822,Z 688.752,A -85,B 0,C 180,E1 2881.877,E2 2881.877} C_VEL
LIN {X 0,Y 47.256,Z 702.755,A -85,B 0,C 180,E1 2869.024,E2 2869.024} C_VEL
LIN {X 0,Y 51.483,Z 717.036,A -85,B 0,C 180,E1 2854.707,E2 2854.707} C_VEL
LIN {X 0,Y 59.86,Z 731.468,A -85,B 0,C 180,E1 2840.602,E2 2840.602} C_VEL
LIN {X 0,Y 63.711,Z 736.155,A -85,B 0,C 180,E1 2836.212,E2 2836.212} C_VEL
LIN {X 0,Y 61.438,Z 735.405,A -85,B 0,C 180,E1 2831.543,E2 2831.543} C_VEL
LIN {X 0,Y 54.602,Z 742.408,A -85,B 0,C 180,E1 2825.872,E2 2825.872} C_VEL
LIN {X 0,Y 48.705,Z 751.718,A -85,B 0,C 180,E1 2815.538,E2 2815.538} C_VEL
LIN {X 0,Y 46.257,Z 762.549,A -85,B 0,C 180,E1 2799.958,E2 2799.958} C_VEL
LIN {X 0,Y 47.979,Z 772.191,A -85,B 0,C 180,E1 2784.019,E2 2784.019} C_VEL
LIN {X 0,Y 49.137,Z 775.285,A -85,B 0,C 180,E1 2778.259,E2 2778.259} C_VEL
LIN {X 0,Y 52.151,Z 782.285,A -85,B 0,C 180,E1 2754.888,E2 2754.888} C_VEL
LIN {X 0,Y 56.738,Z 785.289,A -85,B 0,C 180,E1 2744.112,E2 2744.112} C_VEL
LIN {X 0,Y 47.752,Z 775.715,A -85,B 0,C 180,E1 2724.756,E2 2724.756} C_VEL
LIN {X 0,Y 45.09,Z 769.201,A -85,B 0,C 180,E1 2711.51,E2 2711.51} C_VEL
LIN {X 0,Y 43.71,Z 760.526,A -85,B 0,C 180,E1 2696.063,E2 2696.063} C_VEL
LIN {X 0,Y 45.147,Z 748.195,A -85,B 0,C 180,E1 2677.881,E2 2677.881} C_VEL
LIN {X 0,Y 49.87,Z 733.944,A -85,B 0,C 180,E1 2662.3,E2 2662.3} C_VEL
LIN {X 0,Y 56.946,Z 717.507,A -85,B 0,C 180,E1 2650.2,E2 2650.2} C_VEL
LIN {X 0,Y 65.04,Z 699.153,A -85,B 0,C 180,E1 2641.512,E2 2641.512} C_VEL
LIN {X 0,Y 73.056,Z 679.5,A -85,B 0,C 180,E1 2635.404,E2 2635.404} C_VEL
LIN {X 0,Y 80.27,Z 659,A -85,B 0,C 180,E1 2631.176,E2 2631.176} C_VEL
LIN {X 0,Y 86.002,Z 639.13,A -85,B 0,C 180,E1 2628.385,E2 2628.385} C_VEL
LIN {X 0,Y 87.103,Z 631.675,A -85,B 0,C 180,E1 2627.181,E2 2627.181} C_VEL
LIN {X 0,Y 86.945,Z 611.58,A -85,B 0,C 180,E1 2622.549,E2 2622.549} C_VEL
LIN {X 0,Y 87.906,Z 605.128,A -85,B 0,C 180,E1 2621.624,E2 2621.624} C_VEL
LIN {X 0,Y 104.91,Z 534.223,A -85,B 0,C 180,E1 2616.368,E2 2616.368} C_VEL
LIN {X 0,Y 100.365,Z 519.55,A -85,B 0,C 180,E1 2609.572,E2 2609.572} C_VEL
LIN {X 0,Y 96.536,Z 507.728,A -85,B 0,C 180,E1 2602.636,E2 2602.636} C_VEL
LIN {X 0,Y 94.656,Z 502.486,A -85,B 0,C 180,E1 2598.731,E2 2598.731} C_VEL
LIN {X 0,Y 91.343,Z 504.446,A -85,B 0,C 180,E1 2595.061,E2 2595.061} C_VEL
LIN {X 0,Y 89.499,Z 506.115,A -85,B 0,C 180,E1 2592.935,E2 2592.935} C_VEL
LIN {X 0,Y 84.946,Z 516.683,A -85,B 0,C 180,E1 2590.207,E2 2590.207} C_VEL
LIN {X 0,Y 79.852,Z 530.46,A -85,B 0,C 180,E1 2587.556,E2 2587.556} C_VEL
LIN {X 0,Y 77.039,Z 537.662,A -85,B 0,C 180,E1 2585.637,E2 2585.637} C_VEL
LIN {X 0,Y 73.628,Z 547.402,A -85,B 0,C 180,E1 2583.566,E2 2583.566} C_VEL
LIN {X 0,Y 63.13,Z 580.859,A -85,B 0,C 180,E1 2578.572,E2 2578.572} C_VEL
LIN {X 0,Y 56.835,Z 600.86,A -85,B 0,C 180,E1 2573.263,E2 2573.263} C_VEL
LIN {X 0,Y 53.449,Z 612.093,A -85,B 0,C 180,E1 2568.443,E2 2568.443} C_VEL
LIN {X 0,Y 46.316,Z 638.887,A -85,B 0,C 180,E1 2560.062,E2 2560.062} C_VEL
LIN {X 0,Y 41.937,Z 656.379,A -85,B 0,C 180,E1 2550.84,E2 2550.84} C_VEL
LIN {X 0,Y 38.638,Z 673.105,A -85,B 0,C 180,E1 2537.315,E2 2537.315} C_VEL
LIN {X 0,Y 38.06,Z 690.978,A -85,B 0,C 180,E1 2517.744,E2 2517.744} C_VEL
LIN {X 0,Y 42.515,Z 709.855,A -85,B 0,C 180,E1 2495.699,E2 2495.699} C_VEL
LIN {X 0,Y 50.632,Z 726.257,A -85,B 0,C 180,E1 2479.334,E2 2479.334} C_VEL
LIN {X 0,Y 54.518,Z 732.097,A -85,B 0,C 180,E1 2474.338,E2 2474.338} C_VEL
LIN {X 0,Y 46.583,Z 740.397,A -85,B 0,C 180,E1 2466.941,E2 2466.941} C_VEL
LIN {X 0,Y 40.82,Z 749.813,A -85,B 0,C 180,E1 2454.608,E2 2454.608} C_VEL
LIN {X 0,Y 38.997,Z 760.765,A -85,B 0,C 180,E1 2435.887,E2 2435.887} C_VEL
LIN {X 0,Y 41.805,Z 770.411,A -85,B 0,C 180,E1 2417.57,E2 2417.57} C_VEL
LIN {X 0,Y 42.414,Z 771.624,A -85,B 0,C 180,E1 2414.971,E2 2414.971} C_VEL
LIN {X 0,Y 46.977,Z 778.8,A -85,B 0,C 180,E1 2388.715,E2 2388.715} C_VEL
LIN {X 0,Y 48.37,Z 779.697,A -85,B 0,C 180,E1 2385.111,E2 2385.111} C_VEL
LIN {X 0,Y 40.203,Z 770.484,A -85,B 0,C 180,E1 2365.009,E2 2365.009} C_VEL
LIN {X 0,Y 37.48,Z 763.97,A -85,B 0,C 180,E1 2350.761,E2 2350.761} C_VEL
LIN {X 0,Y 36.274,Z 753.601,A -85,B 0,C 180,E1 2330.478,E2 2330.478} C_VEL
LIN {X 0,Y 39.207,Z 740.062,A -85,B 0,C 180,E1 2309.331,E2 2309.331} C_VEL
LIN {X 0,Y 45.771,Z 724.281,A -85,B 0,C 180,E1 2292.96,E2 2292.96} C_VEL
LIN {X 0,Y 53.732,Z 707.435,A -85,B 0,C 180,E1 2282.146,E2 2282.146} C_VEL
LIN {X 0,Y 62.572,Z 687.933,A -85,B 0,C 180,E1 2274.378,E2 2274.378} C_VEL
LIN {X 0,Y 70.49,Z 668.032,A -85,B 0,C 180,E1 2269.39,E2 2269.39} C_VEL
LIN {X 0,Y 77.463,Z 646.935,A -85,B 0,C 180,E1 2265.923,E2 2265.923} C_VEL
LIN {X 0,Y 84.011,Z 621.581,A -85,B 0,C 180,E1 2263.167,E2 2263.167} C_VEL
LIN {X 0,Y 87.906,Z 605.128,A -85,B 0,C 180,E1 2261.624,E2 2261.624} C_VEL
LIN {X 0,Y 88.981,Z 597.626,A -85,B 0,C 180,E1 2260.516,E2 2260.516} C_VEL
LIN {X 0,Y 89.571,Z 577.581,A -85,B 0,C 180,E1 2255.998,E2 2255.998} C_VEL
LIN {X 0,Y 90.703,Z 571.145,A -85,B 0,C 180,E1 2255.192,E2 2255.192} C_VEL
LIN {X 0,Y 99.234,Z 536.486,A -85,B 0,C 180,E1 2252.953,E2 2252.953} C_VEL
LIN {X 0,Y 95.537,Z 523.41,A -85,B 0,C 180,E1 2246.4,E2 2246.4} C_VEL
LIN {X 0,Y 92.331,Z 512.309,A -85,B 0,C 180,E1 2239.392,E2 2239.392} C_VEL
LIN {X 0,Y 91.891,Z 510.951,A -85,B 0,C 180,E1 2238.322,E2 2238.322} C_VEL
LIN {X 0,Y 90.372,Z 512.163,A -85,B 0,C 180,E1 2236.812,E2 2236.812} C_VEL
LIN {X 0,Y 86.839,Z 520.007,A -85,B 0,C 180,E1 2234.96,E2 2234.96} C_VEL
LIN {X 0,Y 81.416,Z 533.903,A -85,B 0,C 180,E1 2232.571,E2 2232.571} C_VEL
LIN {X 0,Y 78.492,Z 541.067,A -85,B 0,C 180,E1 2230.916,E2 2230.916} C_VEL
LIN {X 0,Y 75.273,Z 549.879,A -85,B 0,C 180,E1 2229.332,E2 2229.332} C_VEL
LIN {X 0,Y 64.184,Z 583.71,A -85,B 0,C 180,E1 2225.288,E2 2225.288} C_VEL
LIN {X 0,Y 57.307,Z 603.766,A -85,B 0,C 180,E1 2220.738,E2 2220.738} C_VEL
LIN {X 0,Y 53.456,Z 614.874,A -85,B 0,C 180,E1 2216.585,E2 2216.585} C_VEL
LIN {X 0,Y 45.533,Z 641.093,A -85,B 0,C 180,E1 2209.618,E2 2209.618} C_VEL
LIN {X 0,Y 39.702,Z 659.162,A -85,B 0,C 180,E1 2200.906,E2 2200.906} C_VEL
LIN {X 0,Y 34.715,Z 675.768,A -85,B 0,C 180,E1 2187.443,E2 2187.443} C_VEL
LIN {X 0,Y 32.021,Z 692.94,A -85,B 0,C 180,E1 2166.277,E2 2166.277} C_VEL
LIN {X 0,Y 34.832,Z 711.839,A -85,B 0,C 180,E1 2138.975,E2 2138.975} C_VEL
LIN {X 0,Y 43.246,Z 729.185,A -85,B 0,C 180,E1 2117.897,E2 2117.897} C_VEL
LIN {X 0,Y 44.801,Z 731.485,A -85,B 0,C 180,E1 2115.575,E2 2115.575} C_VEL
LIN {X 0,Y 36.773,Z 740.86,A -85,B 0,C 180,E1 2104.82,E2 2104.82} C_VEL
LIN {X 0,Y 31.967,Z 751.283,A -85,B 0,C 180,E1 2086.35,E2 2086.35} C_VEL
LIN {X 0,Y 33.957,Z 764.313,A -85,B 0,C 180,E1 2058.106,E2 2058.106} C_VEL
LIN {X 0,Y 35.935,Z 767.797,A -85,B 0,C 180,E1 2050.495,E2 2050.495} C_VEL
LIN {X 0,Y 40.258,Z 773.641,A -85,B 0,C 180,E1 2026.588,E2 2026.588} C_VEL
LIN {X 0,Y 33.039,Z 765.403,A -85,B 0,C 180,E1 2006.994,E2 2006.994} C_VEL
LIN {X 0,Y 29.815,Z 758.192,A -85,B 0,C 180,E1 1989.65,E2 1989.65} C_VEL
LIN {X 0,Y 29.213,Z 746.523,A -85,B 0,C 180,E1 1963.407,E2 1963.407} C_VEL
LIN {X 0,Y 33.653,Z 732.682,A -85,B 0,C 180,E1 1940.297,E2 1940.297} C_VEL
LIN {X 0,Y 41.298,Z 716.952,A -85,B 0,C 180,E1 1924.594,E2 1924.594} C_VEL
LIN {X 0,Y 50.472,Z 698.743,A -85,B 0,C 180,E1 1914.316,E2 1914.316} C_VEL
LIN {X 0,Y 59.359,Z 679.339,A -85,B 0,C 180,E1 1907.877,E2 1907.877} C_VEL
LIN {X 0,Y 67.047,Z 659.684,A -85,B 0,C 180,E1 1903.804,E2 1903.804} C_VEL
LIN {X 0,Y 73.769,Z 638.381,A -85,B 0,C 180,E1 1900.952,E2 1900.952} C_VEL
LIN {X 0,Y 90.703,Z 571.145,A -85,B 0,C 180,E1 1895.192,E2 1895.192} C_VEL
LIN {X 0,Y 91.345,Z 566.111,A -85,B 0,C 180,E1 1894.375,E2 1894.375} C_VEL
LIN {X 0,Y 90.793,Z 553.025,A -85,B 0,C 180,E1 1890.493,E2 1890.493} C_VEL
LIN {X 0,Y 91.456,Z 548.696,A -85,B 0,C 180,E1 1889.872,E2 1889.872} C_VEL
LIN {X 0,Y 93.858,Z 538.845,A -85,B 0,C 180,E1 1889.237,E2 1889.237} C_VEL
LIN {X 0,Y 90.652,Z 526.125,A -85,B 0,C 180,E1 1882.235,E2 1882.235} C_VEL
LIN {X 0,Y 89.598,Z 522.283,A -85,B 0,C 180,E1 1879.61,E2 1879.61} C_VEL
LIN {X 0,Y 83.725,Z 536.8,A -85,B 0,C 180,E1 1877.497,E2 1877.497} C_VEL
LIN {X 0,Y 80.512,Z 544.423,A -85,B 0,C 180,E1 1875.986,E2 1875.986} C_VEL
LIN {X 0,Y 77.56,Z 552.162,A -85,B 0,C 180,E1 1874.854,E2 1874.854} C_VEL
LIN {X 0,Y 66.17,Z 585.939,A -85,B 0,C 180,E1 1871.822,E2 1871.822} C_VEL
LIN {X 0,Y 58.74,Z 606.37,A -85,B 0,C 180,E1 1868.078,E2 1868.078} C_VEL
LIN {X 0,Y 54.44,Z 617.557,A -85,B 0,C 180,E1 1864.611,E2 1864.611} C_VEL
LIN {X 0,Y 45.992,Z 643.055,A -85,B 0,C 180,E1 1859.33,E2 1859.33} C_VEL
LIN {X 0,Y 39.139,Z 660.841,A -85,B 0,C 180,E1 1852.37,E2 1852.37} C_VEL
LIN {X 0,Y 32.346,Z 677.509,A -85,B 0,C 180,E1 1840.479,E2 1840.479} C_VEL
LIN {X 0,Y 26.932,Z 694.74,A -85,B 0,C 180,E1 1818.398,E2 1818.398} C_VEL
LIN {X 0,Y 27.418,Z 714.245,A -85,B 0,C 180,E1 1783.04,E2 1783.04} C_VEL
LIN {X 0,Y 35.146,Z 731.128,A -85,B 0,C 180,E1 1756.843,E2 1756.843} C_VEL
LIN {X 0,Y 27.272,Z 741.281,A -85,B 0,C 180,E1 1740.883,E2 1740.883} C_VEL
LIN {X 0,Y 24.558,Z 752.601,A -85,B 0,C 180,E1 1712.334,E2 1712.334} C_VEL
LIN {X 0,Y 29.73,Z 763.706,A -85,B 0,C 180,E1 1684.074,E2 1684.074} C_VEL
LIN {X 0,Y 32.382,Z 767.081,A -85,B 0,C 180,E1 1668.84,E2 1668.84} C_VEL
LIN {X 0,Y 26.382,Z 760.541,A -85,B 0,C 180,E1 1652.042,E2 1652.042} C_VEL
LIN {X 0,Y 22.113,Z 751.847,A -85,B 0,C 180,E1 1627.793,E2 1627.793} C_VEL
LIN {X 0,Y 22.79,Z 738.94,A -85,B 0,C 180,E1 1592.567,E2 1592.567} C_VEL
LIN {X 0,Y 29.932,Z 723.349,A -85,B 0,C 180,E1 1566.704,E2 1566.704} C_VEL
LIN {X 0,Y 39.578,Z 705.875,A -85,B 0,C 180,E1 1552.759,E2 1552.759} C_VEL
LIN {X 0,Y 48.728,Z 688.17,A -85,B 0,C 180,E1 1545.329,E2 1545.329} C_VEL
LIN {X 0,Y 57.466,Z 668.61,A -85,B 0,C 180,E1 1540.556,E2 1540.556} C_VEL
LIN {X 0,Y 65.042,Z 647.945,A -85,B 0,C 180,E1 1537.456,E2 1537.456} C_VEL
LIN {X 0,Y 72.298,Z 622.481,A -85,B 0,C 180,E1 1535,E2 1535} C_VEL
LIN {X 0,Y 91.456,Z 548.696,A -85,B 0,C 180,E1 1529.872,E2 1529.872} C_VEL
LIN {X 0,Y 90.971,Z 547.911,A -85,B 0,C 180,E1 1529.223,E2 1529.223} C_VEL
LIN {X 0,Y 89.238,Z 548.498,A -85,B 0,C 180,E1 1527.794,E2 1527.794} C_VEL
LIN {X 0,Y 86.006,Z 551.586,A -85,B 0,C 180,E1 1525.564,E2 1525.564} C_VEL
LIN {X 0,Y 79.734,Z 561.147,A -85,B 0,C 180,E1 1521.743,E2 1521.743} C_VEL
LIN {X 0,Y 76.088,Z 568.251,A -85,B 0,C 180,E1 1519.773,E2 1519.773} C_VEL
LIN {X 0,Y 74.151,Z 573.149,A -85,B 0,C 180,E1 1519.116,E2 1519.116} C_VEL
LIN {X 0,Y 64.162,Z 600.824,A -85,B 0,C 180,E1 1516.447,E2 1516.447} C_VEL
LIN {X 0,Y 57.694,Z 616.78,A -85,B 0,C 180,E1 1513.027,E2 1513.027} C_VEL
LIN {X 0,Y 56.124,Z 620.872,A -85,B 0,C 180,E1 1512.181,E2 1512.181} C_VEL
LIN {X 0,Y 47.748,Z 644.609,A -85,B 0,C 180,E1 1508.729,E2 1508.729} C_VEL
LIN {X 0,Y 39.684,Z 663.27,A -85,B 0,C 180,E1 1503.44,E2 1503.44} C_VEL
LIN {X 0,Y 30.665,Z 681.355,A -85,B 0,C 180,E1 1493.025,E2 1493.025} C_VEL
LIN {X 0,Y 22.032,Z 700.179,A -85,B 0,C 180,E1 1468.462,E2 1468.462} C_VEL
LIN {X 0,Y 20.689,Z 719.105,A -85,B 0,C 180,E1 1423.148,E2 1423.148} C_VEL
LIN {X 0,Y 25.812,Z 730.617,A -85,B 0,C 180,E1 1398.817,E2 1398.817} C_VEL
LIN {X 0,Y 18.244,Z 741.642,A -85,B 0,C 180,E1 1372.56,E2 1372.56} C_VEL
LIN {X 0,Y 19.862,Z 753.815,A -85,B 0,C 180,E1 1329.367,E2 1329.367} C_VEL
LIN {X 0,Y 24.715,Z 759.976,A -85,B 0,C 180,E1 1312.681,E2 1312.681} C_VEL
LIN {X 0,Y 18.768,Z 753.664,A -85,B 0,C 180,E1 1295.87,E2 1295.87} C_VEL
LIN {X 0,Y 14.16,Z 742.008,A -85,B 0,C 180,E1 1251.876,E2 1251.876} C_VEL
LIN {X 0,Y 19.432,Z 727.533,A -85,B 0,C 180,E1 1208.13,E2 1208.13} C_VEL
LIN {X 0,Y 29.592,Z 710.787,A -85,B 0,C 180,E1 1188.893,E2 1188.893} C_VEL
LIN {X 0,Y 39.652,Z 693.327,A -85,B 0,C 180,E1 1180.435,E2 1180.435} C_VEL
LIN {X 0,Y 49.714,Z 672.936,A -85,B 0,C 180,E1 1175.383,E2 1175.383} C_VEL
LIN {X 0,Y 57.8,Z 652.971,A -85,B 0,C 180,E1 1172.532,E2 1172.532} C_VEL
LIN {X 0,Y 65.026,Z 629.967,A -85,B 0,C 180,E1 1170.509,E2 1170.509} C_VEL
LIN {X 0,Y 88.804,Z 541.236,A -85,B 0,C 180,E1 1165.156,E2 1165.156} C_VEL
LIN {X 0,Y 87.72,Z 536.981,A -85,B 0,C 180,E1 1162.598,E2 1162.598} C_VEL
LIN {X 0,Y 83.117,Z 547.498,A -85,B 0,C 180,E1 1160.846,E2 1160.846} C_VEL
LIN {X 0,Y 80.387,Z 554.533,A -85,B 0,C 180,E1 1160.048,E2 1160.048} C_VEL
LIN {X 0,Y 74.151,Z 573.149,A -85,B 0,C 180,E1 1159.116,E2 1159.116} C_VEL
LIN {X 0,Y 71.823,Z 581.241,A -85,B 0,C 180,E1 1159.264,E2 1159.264} C_VEL
LIN {X 0,Y 67.475,Z 601.064,A -85,B 0,C 180,E1 1161.791,E2 1161.791} C_VEL
LIN {X 0,Y 64.954,Z 609.01,A -85,B 0,C 180,E1 1161.778,E2 1161.778} C_VEL
LIN {X 0,Y 64.512,Z 610.106,A -85,B 0,C 180,E1 1161.639,E2 1161.639} C_VEL
LIN {X 0,Y 59.14,Z 622.694,A -85,B 0,C 180,E1 1159.332,E2 1159.332} C_VEL
LIN {X 0,Y 50.721,Z 645.716,A -85,B 0,C 180,E1 1157.374,E2 1157.374} C_VEL
LIN {X 0,Y 42.079,Z 664.434,A -85,B 0,C 180,E1 1154.232,E2 1154.232} C_VEL
LIN {X 0,Y 31.862,Z 682.687,A -85,B 0,C 180,E1 1147.787,E2 1147.787} C_VEL
LIN {X 0,Y 20.164,Z 701.61,A -85,B 0,C 180,E1 1130.232,E2 1130.232} C_VEL
LIN {X 0,Y 13.334,Z 720.043,A -85,B 0,C 180,E1 1077.857,E2 1077.857} C_VEL
LIN {X 0,Y 16.518,Z 730.276,A -85,B 0,C 180,E1 1041.901,E2 1041.901} C_VEL
LIN {X 0,Y 10.477,Z 741.921,A -85,B 0,C 180,E1 990.001,E2 990.001} C_VEL
LIN {X 0,Y 13.963,Z 748.941,A -85,B 0,C 180,E1 954.563,E2 954.563} C_VEL
LIN {X 0,Y 6.939,Z 737.195,A -85,B 0,C 180,E1 891.705,E2 891.705} C_VEL
LIN {X 0,Y 14.813,Z 722.346,A -85,B 0,C 180,E1 829.079,E2 829.079} C_VEL
LIN {X 0,Y 26.608,Z 705.109,A -85,B 0,C 180,E1 815.211,E2 815.211} C_VEL
LIN {X 0,Y 37.496,Z 686.589,A -85,B 0,C 180,E1 810,E2 810} C_VEL
LIN {X 0,Y 47.05,Z 666.97,A -85,B 0,C 180,E1 807.221,E2 807.221} C_VEL
LIN {X 0,Y 55.418,Z 645.482,A -85,B 0,C 180,E1 805.458,E2 805.458} C_VEL
LIN {X 0,Y 65.014,Z 613.099,A -85,B 0,C 180,E1 803.667,E2 803.667} C_VEL
LIN {X 0,Y 68.861,Z 599.183,A -85,B 0,C 180,E1 802.916,E2 802.916} C_VEL
LIN {X 0,Y 64.512,Z 610.106,A -85,B 0,C 180,E1 801.639,E2 801.639} C_VEL
LIN {X 0,Y 64.349,Z 610.926,A -85,B 0,C 180,E1 801.581,E2 801.581} C_VEL
LIN {X 0,Y 64.349,Z 706.847,A -85,B 0,C 180,E1 801.581,E2 801.581} C_VEL
LIN {X 0,Y 36.181,Z 706.847,A -85,B 0,C 180,E1 801.216,E2 801.216} C_VEL
LIN {X 0,Y 34.181,Z 704.847,A -85,B 0,C 180,E1 801.167,E2 801.167} C_VEL
LIN {X 0,Y 34.181,Z 691.247,A -85,B 0,C 180,E1 801.167,E2 801.167} C_VEL
LIN {X 0,Y 30.818,Z 689.986,A -85,B 0,C 180,E1 799.146,E2 799.146} C_VEL
LIN {X 0,Y 18.198,Z 707.164,A -85,B 0,C 180,E1 789.085,E2 789.085} C_VEL
LIN {X 0,Y 6.779,Z 725.074,A -85,B 0,C 180,E1 728.493,E2 728.493} C_VEL
LIN {X 0,Y 7.375,Z 729.94,A -85,B 0,C 180,E1 691.191,E2 691.191} C_VEL
LIN {X 0,Y 3.505,Z 735.833,A -85,B 0,C 180,E1 626.575,E2 626.575} C_VEL
LIN {X 0,Y 9.652,Z 720.976,A -85,B 0,C 180,E1 799.8,E2 799.8} C_VEL
LIN {X 0,Y 22.093,Z 704.054,A -85,B 0,C 180,E1 799.57,E2 799.57} C_VEL
LIN {X 0,Y 30.818,Z 689.986,A -85,B 0,C 180,E1 799.146,E2 799.146} C_VEL
LIN {X 0,Y 34.539,Z 691.002,A -85,B 0,C 180,E1 798.922,E2 798.922} C_VEL
LIN {X 0,Y 34.539,Z 855,A -85,B 0,C 180,E1 798.922,E2 798.922} C_VEL
LIN {X 0,Y 34.539,Z 855,A -85,B 0,C 180,E1 798.922,E2 798.922}

QRS_NEXT_CUT()

QRS_NEXT()
QRS_HOME()

END
